// TIA Portal V19 export
DATA_BLOCK "nextDB"   // DB222
{ S7_Optimized_Access := 'TRUE' }
// stored: AutoNumber false, MemoryReserve 100
   VAR
      data : Array[1..100] of Byte;
   END_VAR
BEGIN
END_DATA_BLOCK
